SUBAPPLICATION AbstTwoStateCtrlOneSens (* Subapplication Type *)
  (* Standard: 61499-2 *)
  (* Version 1.0, 2020-07-20, AK120569 *)
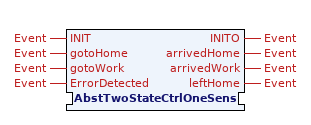
  EVENT_INPUT
    INIT; (* Initialization Request *)
    gotoHome;
    gotoWork;
    ErrorDetected;
  END_EVENT
  EVENT_OUTPUT
    INITO; (* Initialization Confirm *)
    arrivedHome;
    arrivedWork;
    leftHome;
  END_EVENT
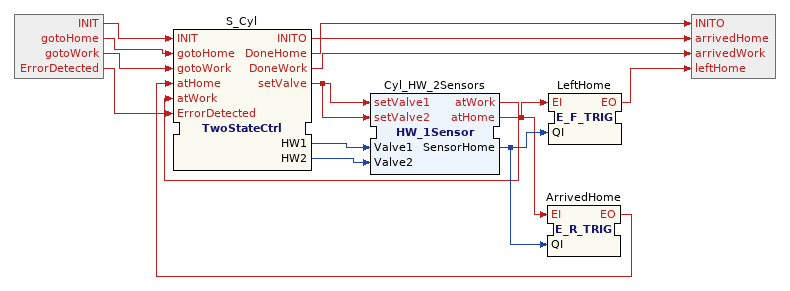
  FBS
    S_Cyl : TwoStateCtrl;
    LeftHome : E_F_TRIG;
    ArrivedHome : E_R_TRIG;
  END_FBS
  SUBAPPS
    Cyl_HW_2Sensors : HW_1Sensor;
  END_SUBAPPS
  EVENT_CONNECTIONS
    INIT TO S_Cyl.INIT;
    gotoHome TO S_Cyl.gotoHome;
    gotoWork TO S_Cyl.gotoWork;
    S_Cyl.INITO TO INITO;
    S_Cyl.DoneHome TO arrivedHome;
    S_Cyl.DoneWork TO arrivedWork;
    S_Cyl.setValve TO Cyl_HW_2Sensors.setValve1;
    S_Cyl.setValve TO Cyl_HW_2Sensors.setValve2;
    Cyl_HW_2Sensors.atWork TO S_Cyl.atWork;
    Cyl_HW_2Sensors.atHome TO LeftHome.EI;
    Cyl_HW_2Sensors.atHome TO ArrivedHome.EI;
    ArrivedHome.EO TO S_Cyl.atHome;
    LeftHome.EO TO leftHome;
    ErrorDetected TO S_Cyl.ErrorDetected;
  END_CONNECTIONS
  DATA_CONNECTIONS
    S_Cyl.HW1 TO Cyl_HW_2Sensors.Valve1;
    S_Cyl.HW2 TO Cyl_HW_2Sensors.Valve2;
    Cyl_HW_2Sensors.SensorHome TO LeftHome.QI;
    Cyl_HW_2Sensors.SensorHome TO ArrivedHome.QI;
  END_CONNECTIONS
END_SUBAPPLICATION
